# EPICS substitutions: testioApp/Db/output.substitutions
file ../../db/output.db {
    pattern     {Sys,           Key    }
                {"BBB01",       "ONOFF" }
}
